PROGRAM MAIN
VAR
END_VAR

END_PROGRAM

(* stored: Version 1.1.0.1
   POU MAIN: Id {061633ad-b962-4bb3-94b7-93cb3f1ee577} *)
